// TIA Portal V17 export
// export: Created 2022-07-20T06:59:40.3494529Z, ExportSetting WithDefaults, DisplayName Totally Integrated Automation Portal, DisplayVersion V17, DisplayName TIA Portal Openness, DisplayVersion V17, DisplayName TIA Portal Version Control Interface, DisplayVersion V17, DisplayName SINAMICS Startdrive Advanced, DisplayVersion V17, DisplayName SINAMICS Startdrive G130, G150, S120, S150, SINAMICS MV, S210, DisplayVersion V17, DisplayName SINAMICS Startdrive G110M, G120, G120C, G120D, G120P, G115D, DisplayVersion V17, DisplayName STEP 7 Professional, DisplayVersion V17, DisplayName STEP 7 Safety, DisplayVersion V17, DisplayName WinCC Advanced, DisplayVersion V17
FUNCTION "FC10011_DintTo2Int" : Void   // FC10011, LAD
TITLE = FC10011_DintTo2Int
{ S7_Optimized_Access := 'TRUE' }
AUTHOR : Anirouddh
FAMILY : 1001x_CONVERT
VERSION : 1.0
// Release note : 
// 1.0 - Feature developped
// stored: AutoNumber false, IsIECCheckEnabled false, SetENOAutomatically false, UDAEnableTagReadback false
   VAR_INPUT
      Dint_Input : DInt;
   END_VAR
   VAR_OUTPUT
      Int_LowWeight : Int;
      Int_HighWeight : Int;
   END_VAR
   VAR_TEMP
      Val_temp1 : DWord;
      Val_temp2 : DWord;
   END_VAR
BEGIN

REGION Network 1 (SCL)
   //Entier bits de poids faibes
   #Val_temp2 := DINT_TO_DWORD(#Dint_Input);
   #Val_temp2 := SHL_DWORD(IN := #Val_temp2, N := 16);
   #Val_temp2 := SHR_DWORD(IN := #Val_temp2, N := 16);
   #Int_LowWeight := DWORD_TO_INT(#Val_temp2);

   //Entier bits de poids ford
   #Val_temp1 := DINT_TO_DWORD(#Dint_Input);
   #Val_temp1 := SHR_DWORD(IN := #Val_temp1, N := 16);
   #Int_HighWeight := DWORD_TO_INT(#Val_temp1);
END_REGION
END_FUNCTION
